FUNCTION_BLOCK SENSOR_DRIVER_SINGLE_PHASE (* Extracted Composite Function Block Type *)
  (* Standard: 61499-2 *)
  (* Version 4/28/2023, Dmitrii *)
  PACKAGE UAO.Hackathon;
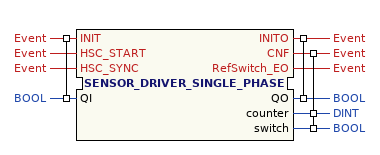
  EVENT_INPUT
    INIT WITH QI; (* Initializes the symbolic link data destination FB with N (1 <= N <= 16) variables *)
    HSC_START; (* Triggers cyclic reading (polling) *)
    HSC_SYNC; (* Synchronization *)
  END_EVENT
  EVENT_OUTPUT
    INITO WITH QO; (* Initialization confirm *)
    CNF WITH counter, switch; (* Execution Confirmation *)
    RefSwitch_EO; (* Event Output *)
  END_EVENT
  VAR_INPUT
    QI : BOOL; (* INIT event input qualifier *)
  END_VAR
  VAR_OUTPUT
    QO : BOOL; (* Output event qualifier *)
    counter : DINT; (* Result: IN1 - IN2 - IN3 - ... *)
    switch : BOOL; (* Current value(i) in the named variable array element *)
  END_VAR
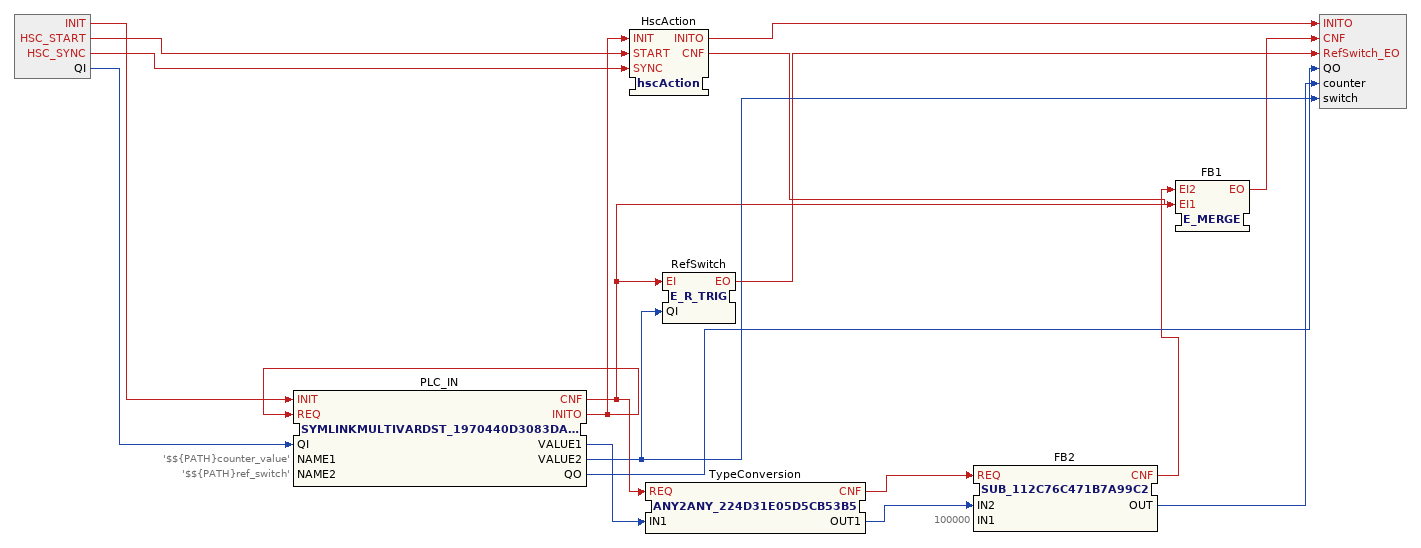
  FBS
    PLC_IN : SYMLINKMULTIVARDST_1970440D3083DA789(NAME1 := '$${PATH}counter_value', NAME2 := '$${PATH}ref_switch'); {SET_ATTRIBUTE(Configuration.GenericFBType.InterfaceParams, Runtime.System#I:=2;VALUE${I$}:DWORD,BOOL)}
    FB2 : SUB_112C76C471B7A99C2(IN1 := 100000); {SET_ATTRIBUTE(Configuration.GenericFBType.InterfaceParams, Runtime.Standard#CNT:=2;IN${CNT$}:DINT)}
    TypeConversion : ANY2ANY_224D31E05D5CB53B5; {SET_ATTRIBUTE(Configuration.GenericFBType.InterfaceParams, Runtime.Standard#CNT:=1;IN${CNT$}:DWORD;OUT${CNT$}:DINT)}
    RefSwitch : E_R_TRIG;
    HscAction : hscAction;
    FB1 : E_MERGE;
  END_FBS
  EVENT_CONNECTIONS
    PLC_IN.CNF TO TypeConversion.REQ;
    TypeConversion.CNF TO FB2.REQ;
    PLC_IN.CNF TO RefSwitch.EI;
    INIT TO PLC_IN.INIT;
    PLC_IN.INITO TO HscAction.INIT;
    FB2.CNF TO FB1.EI2;
    RefSwitch.EO TO RefSwitch_EO;
    HscAction.INITO TO INITO;
    HSC_START TO HscAction.START;
    HSC_SYNC TO HscAction.SYNC;
    PLC_IN.CNF TO FB1.EI1;
    FB1.EO TO CNF;
    HscAction.CNF TO FB1.EI1;
    PLC_IN.INITO TO PLC_IN.REQ;
  END_CONNECTIONS
  DATA_CONNECTIONS
    PLC_IN.VALUE1 TO TypeConversion.IN1;
    TypeConversion.OUT1 TO FB2.IN2;
    PLC_IN.VALUE2 TO RefSwitch.QI;
    QI TO PLC_IN.QI;
    PLC_IN.QO TO QO;
    FB2.OUT TO counter;
    PLC_IN.VALUE2 TO switch;
  END_CONNECTIONS
END_FUNCTION_BLOCK
